% RSLogix 500 project SOLISPLC_ML1100_BAK018.RSS, saved by version 11.00.00.00 %
PROJECT "SOLISPLC"    % processor: Bul.1763 MicroLogix 1100 Series B %

PROGRAM FILES
  LAD 2   4 rungs

DATA FILES
  O0 OUTPUT  4 elements
  I1 INPUT  7 elements
  S2 STATUS  66 elements
  B3 BINARY  1 elements
  T4 TIMER  1 elements
  C5 COUNTER  1 elements
  R6 CONTROL  1 elements
  N7 INTEGER  10 elements
  F8 FLOAT  1 elements
  L9 LONG  10 elements  % long %
  N10 PROD_DATA1  10 elements  % PROD_DATA1 %
  B11 PROD_DATA2  2 elements  % PROD_DATA2 %
  B12 MYBINARY1  10 elements
  N13   12 elements
  F14 FLOAT  10 elements
  F15 MYFLOAT  10 elements

LADDER 2
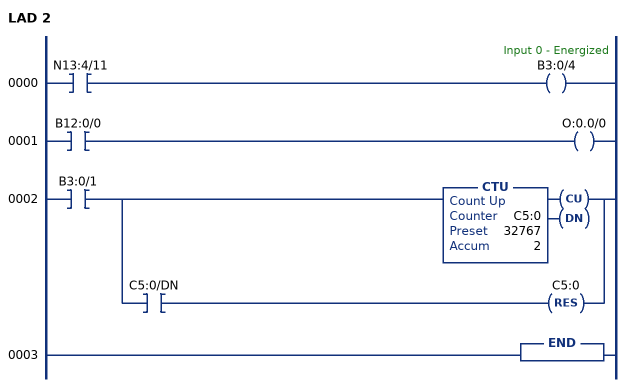
% Rung: 0 %
SOR XIC N13:4/11 OTE B3:0/4 EOR
%   B3:0/4  "Input 0 - Energized" %
% Rung: 1 %
SOR XIC B12:0/0 OTE O:0.0/0 EOR
% Rung: 2 %
SOR XIC B3:0/1 BST CTU C5:0 32767 2 NXB XIC C5:0/DN RES C5:0 BND EOR
% Rung: 3 %
SOR END EOR

DATA TABLE (non-zero values as saved)
DATA T4
% .PRE .ACC %
% T4:0 % 10 7
DATA C5
% .PRE .ACC %
% C5:0 % 32767 2
DATA L9
% L9:0 % 34298 34447 0 0 0
DATA B11
% B11:0 % 0X0040 0X0400
DATA N13
% N13:0 % 0 -234 24 213 0 24234 43 0 0 0
% N13:10 % 0 3452
DATA F15
% F15:0 % 45.4646 46.45646 4.654564e+08 56756.57 567.55
% F15:5 % -34.22 4.3 0 0 0
